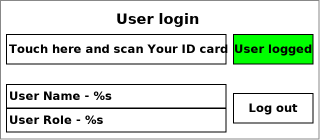
VISUALIZATION vPIM_UserLogin  // 320x140
VAR_IN_OUT
	fbPIM:fbPIM_UserLogin;
END_VAR
    Rectangle (6,34 220x30), "Touch here and scan Your ID card"
        OnMouseClick: write fbPIM.sScanedId via Edit, format %s, password
    Rectangle (6,84 220x24), "User Name - %s", text variable: fbPIM.sUserName, invisible if: NOT fbPIM.bUserLogged
    Rectangle (6,108 220x24), "User Role - %s", text variable: TO_STRING(fbPIM.nUserRole), invisible if: NOT fbPIM.bUserLogged
    RoundedRectangle (233,93 80x30), "Log out", invisible if: NOT fbPIM.bUserLogged
        OnMouseClick: execute { fbPIM.bUserLogged := FALSE; }
    Label (3,4 310x30), "User login"
    Rectangle (233,34 80x30), "DataBase Error", text variable: fbPIM.sUserName, invisible if: NOT fbPIM.bSqlError
    Rectangle (233,34 80x30), "User logged", text variable: fbPIM.sUserName, invisible if: NOT fbPIM.bUserLogged
END_VISUALIZATION

(* stored: Version 1.1.0.1, ProductVersion 3.1.4024.12
   Visu vPIM_UserLogin: Id {2b552e48-e604-43a1-aec8-584fde6d18c7} *)
